SUBAPPLICATION Speedcontrol (* Subapplication Type *)
  (* Standard: 61499-2 *)
  (* Version 1.0, 2026-03-10, 04jul *)
  IMPORT logiBUS::io::DO_LED::LED_FREQ::LED_5HZ;
  IMPORT logiBUS::io::DQ::logiBUS_DO::Output_Q4;
  IMPORT logiBUS::io::DQ::logiBUS_DO::Output_Q5;
  IMPORT logiBUS::io::PI::logiBUS_PI::PulseInput_I2;
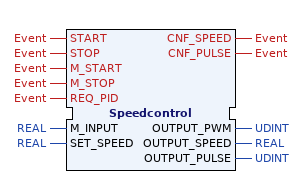
  EVENT_INPUT
    START;
    STOP;
    M_START;
    M_STOP;
    REQ_PID;
  END_EVENT
  EVENT_OUTPUT
    CNF_SPEED;
    CNF_PULSE;
  END_EVENT
  VAR_INPUT
    M_INPUT : REAL;
    SET_SPEED : REAL;
  END_VAR
  VAR_OUTPUT
    OUTPUT_PWM : UDINT;
    OUTPUT_SPEED : REAL;
    OUTPUT_PULSE : UDINT;
  END_VAR
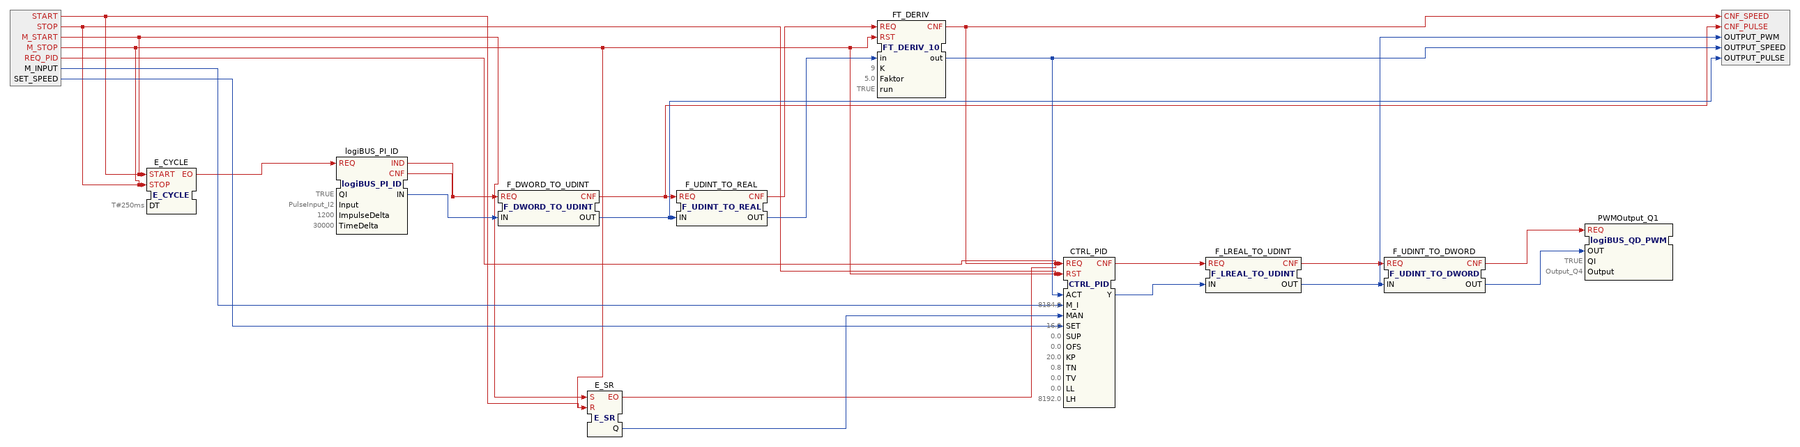
  FBS
    logiBUS_PI_ID : logiBUS::io::PI::logiBUS_PI_ID(QI := TRUE, Input := PulseInput_I2, ImpulseDelta := 1200, TimeDelta := 30000);
    FT_DERIV : OSCAT::Basic::POUs::Engineering::Control::FT_DERIV_10(K := 9, Faktor := 5.0, run := TRUE);
    F_DWORD_TO_UDINT : iec61131::conversion::F_DWORD_TO_UDINT;
    F_UDINT_TO_REAL : iec61131::conversion::F_UDINT_TO_REAL;
    PWMOutput_Q1 : logiBUS::io::DQ::logiBUS_QD_PWM(QI := TRUE, Output := Output_Q4);
    CTRL_PID : OSCAT::Basic::POUs::Engineering::Control::CTRL_PID(SET := 16.0, SUP := 0.0, OFS := 0.0, M_I := 8184.0, KP := 20.0, TN := 0.8, TV := 0.0, LL := 0.0, LH := 8192.0);
    F_LREAL_TO_UDINT : iec61131::conversion::F_LREAL_TO_UDINT;
    F_UDINT_TO_DWORD : iec61131::conversion::F_UDINT_TO_DWORD;
    E_CYCLE : iec61499::events::E_CYCLE(DT := T#250ms);
    E_SR : iec61499::events::E_SR;
  END_FBS
  EVENT_CONNECTIONS
    F_DWORD_TO_UDINT.CNF TO F_UDINT_TO_REAL.REQ;
    F_UDINT_TO_REAL.CNF TO FT_DERIV.REQ;
    FT_DERIV.CNF TO CTRL_PID.REQ;
    CTRL_PID.CNF TO F_LREAL_TO_UDINT.REQ;
    F_LREAL_TO_UDINT.CNF TO F_UDINT_TO_DWORD.REQ;
    F_UDINT_TO_DWORD.CNF TO PWMOutput_Q1.REQ;
    E_CYCLE.EO TO logiBUS_PI_ID.REQ;
    START TO E_CYCLE.START;
    E_SR.EO TO CTRL_PID.REQ;
    M_START TO E_SR.S;
    M_STOP TO E_SR.R;
    START TO E_SR.R;
    M_STOP TO CTRL_PID.RST;
    STOP TO CTRL_PID.RST;
    REQ_PID TO CTRL_PID.REQ;
    FT_DERIV.CNF TO CNF_SPEED;
    M_START TO E_CYCLE.START;
    STOP TO E_CYCLE.STOP;
    M_STOP TO E_CYCLE.STOP;
    logiBUS_PI_ID.IND TO F_DWORD_TO_UDINT.REQ;
    logiBUS_PI_ID.CNF TO F_DWORD_TO_UDINT.REQ;
    M_STOP TO FT_DERIV.RST;
    F_DWORD_TO_UDINT.CNF TO CNF_PULSE;
  END_CONNECTIONS
  DATA_CONNECTIONS
    logiBUS_PI_ID.IN TO F_DWORD_TO_UDINT.IN;
    F_DWORD_TO_UDINT.OUT TO F_UDINT_TO_REAL.IN;
    F_UDINT_TO_REAL.OUT TO FT_DERIV.in;
    FT_DERIV.out TO CTRL_PID.ACT;
    CTRL_PID.Y TO F_LREAL_TO_UDINT.IN;
    F_LREAL_TO_UDINT.OUT TO F_UDINT_TO_DWORD.IN;
    F_UDINT_TO_DWORD.OUT TO PWMOutput_Q1.OUT;
    M_INPUT TO CTRL_PID.M_I;
    F_LREAL_TO_UDINT.OUT TO OUTPUT_PWM;
    E_SR.Q TO CTRL_PID.MAN;
    SET_SPEED TO CTRL_PID.SET;
    FT_DERIV.out TO OUTPUT_SPEED;
    F_DWORD_TO_UDINT.OUT TO OUTPUT_PULSE;
  END_CONNECTIONS
END_SUBAPPLICATION
